(* PLC project  *)

PROGRAM P
  VAR
    tmr : TON;
  END_VAR

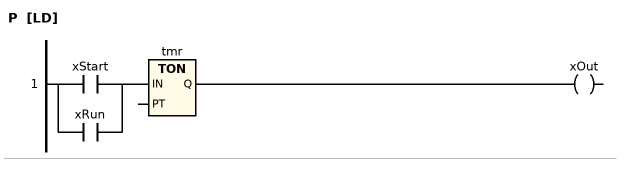
(* LD diagram, written out as Structured Text *)
tmr(IN := xStart OR xRun);
xOut := tmr.Q;
END_PROGRAM
